// TIA Portal V17 export
// export: Created 2022-03-12T16:05:35.5808644Z, ExportSetting WithDefaults, DisplayName Totally Integrated Automation Portal, DisplayVersion V17, DisplayName TIA Portal Openness, DisplayVersion V17, DisplayName TIA Portal Version Control Interface, DisplayVersion V17, DisplayName STEP 7 Professional, DisplayVersion V17, DisplayName STEP 7 Safety, DisplayVersion V17, DisplayName WinCC Advanced / Unified PC, DisplayVersion V17
TYPE "typeLPMLV30_NamesConfiguration"
TITLE = typeLPMLV30_NamesConfiguration
// Support: tech.team.motioncontrol@siemens.com 
// Fax: +49 (0) 9131/98-1297
// stored: IsFailsafeCompliant false
   STRUCT
      unitModesNames : Array[0.."LPMLV30_LANGUAGES_UPPER_LIM", 0.."LPMLV30_MODES_UPPER_LIM"] of String[18];   // Names of unit modes [First index language, Second unit mode no]
      statesNames : Array[0.."LPMLV30_LANGUAGES_UPPER_LIM", 0.."LPMLV30_STATES_UPPER_LIM"] of String[16];   // Names of states [First index language, Second state no]
   END_STRUCT;
   // unitModesNames[0,0] := 'Invalid';
   // unitModesNames[0,1] := 'Production';
   // unitModesNames[0,2] := 'Maintenance';
   // unitModesNames[0,3] := 'Manual';
   // unitModesNames[0,4] := 'User Mode 01';
   // unitModesNames[1,0] := 'Undefiniert';
   // unitModesNames[1,1] := 'Produktion';
   // unitModesNames[1,2] := 'Wartung';
   // unitModesNames[1,3] := 'Hand';
   // unitModesNames[1,4] := 'Benutzer Mode 01';
   // statesNames[0,0] := 'Undefined';
   // statesNames[0,1] := 'Clearing';
   // statesNames[0,2] := 'Stopped';
   // statesNames[0,3] := 'Starting';
   // statesNames[0,4] := 'Idle';
   // statesNames[0,5] := 'Suspended';
   // statesNames[0,6] := 'Execute';
   // statesNames[0,7] := 'Stopping';
   // statesNames[0,8] := 'Aborting';
   // statesNames[0,9] := 'Aborted';
   // statesNames[0,10] := 'Holding';
   // statesNames[0,11] := 'Held';
   // statesNames[0,12] := 'UnHolding';
   // statesNames[0,13] := 'Suspending';
   // statesNames[0,14] := 'UnSuspending';
   // statesNames[0,15] := 'Resetting';
   // statesNames[0,16] := 'Completing';
   // statesNames[0,17] := 'Complete';
   // statesNames[1,0] := 'Undefiniert';
   // statesNames[1,1] := 'Clearing';
   // statesNames[1,2] := 'Stopped';
   // statesNames[1,3] := 'Starting';
   // statesNames[1,4] := 'Idle';
   // statesNames[1,5] := 'Suspended';
   // statesNames[1,6] := 'Execute';
   // statesNames[1,7] := 'Stopping';
   // statesNames[1,8] := 'Aborting';
   // statesNames[1,9] := 'Aborted';
   // statesNames[1,10] := 'Holding';
   // statesNames[1,11] := 'Held';
   // statesNames[1,12] := 'UnHolding';
   // statesNames[1,13] := 'Suspending';
   // statesNames[1,14] := 'UnSuspending';
   // statesNames[1,15] := 'Resetting';
   // statesNames[1,16] := 'Completing';
   // statesNames[1,17] := 'Complete';
END_TYPE
